Fanuc KAREL source: kt00440.KL

-- PROVISIONAL review KL for V1013-1; original PC SHA256 74c1192c9b50b48410a0b2e46b6ca814c01d949926506658eff7fa85ed2d4386
-- Incomplete behavior may be omitted. Consult companion uncertainty JSON. Do not deploy.
PROGRAM KT00440
%NOLOCKGROUP
VAR
  I1 : INTEGER
  OUT : BOOLEAN
-- UNRESOLVED_DECL H2 type=002017
BEGIN
  -- UNRESOLVED_PC offsets 5-16; opcodes 2E,23
  -- UNRESOLVED_PC offsets 21-35; opcodes 2E,22,9D,33,B4
  -- UNRESOLVED_PC offsets 40-62; opcodes 21,22,9D,33,B3,5C,23
  -- UNRESOLVED_PC offsets 67-71; opcodes 7F
END KT00440
